(* PLC project CoDeSys External Library Template, WAGO e!COCKPIT e!COCKPIT, author 3S - Smart Software Solutions GmbH *)
(* stored: creationDateTime 2019-10-29T12:37:19.528471, version 3.5.5.30, modificationDateTime 2019-10-29T12:36:39.3744516, organization 3S - Smart Software Solutions GmbH *)
(* Library project template with all possible element types, docu and a sample project structure *)

TYPE typHarmonogramJSON : STRUCT
  sPokoj : STRING(3);
  sPietro : STRING(2);
  arHarmonogramTygodniowy : ARRAY[0..6] OF typHarmonogramDzien;
  arWyjatki : ARRAY[0..24] OF typHarmonogramWyjatek;
END_STRUCT;
END_TYPE
